{attribute 'qualified_only'}
VAR_GLOBAL
	Q1 AT %Q*: BOOL;	// Linearantrieb Rechtslauf
	Q2 AT %Q*: BOOL;	// Linearantrieb Linkslauf
	P1 AT %Q*: BOOL;	// Meldeleuchte im Taster S1 (weiß)
	P2 AT %Q*: BOOL;	// Meldeleuchte weiß
	P3 AT %Q*: BOOL;	// Meldeleuchte rot
	P4 AT %Q*: BOOL;	// Meldeleuchte grün
END_VAR

(* stored: Version 1.1.0.1, ProductVersion 3.1.4024.5
   GVL DA: Id {efa3d63a-96e1-4204-b1e7-9f3703bd4f03} *)
